         CALL  #MOV_Descarga
         ( Sensor_Pieza               := ,
           Sensor_Pinza_Llena         := ,
           Sensor_Llegada_a_Maquina   := ,
           Sensor_Llegada_a_Buffer    := ,
           "Sensor_Llegada_a _Reposo" := ,
           EMER                       := TRUE,
           Tiempo_lim                 := #Tiempo_lim,
           Timer_LIM                  := #Timer_LIM,
           MOV1                       := #Mov1,
           MOV2                       := #Mov2,
           MOV3                       := #Mov3,
           ACT1                       := #Act1,
           ACT2                       := #Act2,
           Aviso_Error_Tiempo_Limite  := #Aviso_Tiempo_Lim,
           Aviso_Fin_Maniobra         := #Aviso_Fin_Maniobra,
           Aviso_Error_No_Pieza       := #Aviso_No_Pieza,
           Aviso_Error_Pinza_Abierta  := #Aviso_Pinza_Abierta
         );



   _ERROR_ASINCRONO:NOP   0;
END_REGION

REGION Network 6: SALIDA ERROR SINCRONO
         A     #X_Error_Sincrono;
         AN    #Aviso_Error_Sincrono;
         S     #X_REPOSO;
         R     #X_Error_Sincrono;
END_REGION

REGION Network 7: SALIDA ERROR ASINCRONO
         A     #X_Error_Asincrono;
         AN    #Aviso_Error_Asincrono;
         S     #X_REPOSO;
         R     #X_Error_Asincrono;
END_REGION

REGION Network 8: START===TRUE
         A     #START;
         FP    #BDT;

         S     #X_REPOSO;
         R     #X_1_1;
         R     #X_1_2;
END_REGION

REGION Network 9: X_REPOSO--->X_1_1
   // Este modo se activa para el torno y la prensa
         A     #X_REPOSO;
         A     #X_Marcha_1;
         AN    #X_Marcha_2;
         A     #Sensor_Llegada_a_Reposo;
         A     #Sensor_Pieza;
         AN    #Sensor_Pinza_Llena;
         AN    #Sensor_Llegada_Carga;
         AN    #Sensor_Llegada_Descarga;


         S     #X_1_1;
         R     #X_REPOSO;
END_REGION

REGION Network 10: X_REPOSO--->X_1_2
   // Este modo se activa
         A     #X_REPOSO;
         A     #X_Marcha_2;
         AN    #X_Marcha_1;
         A     #Sensor_Llegada_a_Reposo;
         A     #Sensor_Pieza;  //si no hay pieza no llamo al bloque  NO UTILITY
         AN    #Sensor_Pinza_Llena;  //la pinza esta ocupada, no puede ir a por otra pieza
         AN    #Sensor_Llegada_Carga;
         AN    #Sensor_Llegada_Descarga;


         S     #X_1_2;
         R     #X_REPOSO;
END_REGION

REGION Network 11: X_1_1--->X_REPOSO
         A     #X_1_1;
         A     #Aviso_Fin_Maniobra;

         S     #X_REPOSO;
         R     #X_1_1;
         R     #Aviso_Fin_Maniobra;
END_REGION

REGION Network 12: X_1_2--->X_REPOSO
         A     #X_1_2;
         A     #Aviso_Fin_Maniobra;

         S     #X_REPOSO;
         R     #X_1_2;
         R     #Aviso_Fin_Maniobra;
END_REGION

REGION Network 13: TRAT X_REPOSO
         A     #X_REPOSO;
         =     #STDBY;
END_REGION

REGION Network 14: TRAT X_1_1
         A     #X_1_1;


         JCN   _MOV_1;

         CALL  #MOV_Carga
         ( Sensor_Pieza               := #Sensor_Pieza,
           Sensor_Pinza_Llena         := #Sensor_Pinza_Llena,
           Sensor_Llegada_a_Buffer    := #Sensor_Llegada_Carga,
           Sensor_Llegada_a_Maquina   := #Sensor_Llegada_Descarga,
           "Sensor_Llegada_a _Reposo" := #Sensor_Llegada_a_Reposo,
           EMER                       := FALSE,
           Tiempo_lim                 := #Tiempo_lim,
           Timer_LIM                  := #Timer_LIM,
           MOV1                       := #Mov1,
           MOV2                       := #Mov2,
           MOV3                       := #Mov3,
           ACT1                       := #Act1,
           ACT2                       := #Act2,
           WAIT1                      := #Wait,
           Aviso_Error_Tiempo_Limite  := #Aviso_Tiempo_Lim,
           Aviso_Fin_Maniobra         := #Aviso_Fin_Maniobra,
           Aviso_Error_No_Pieza       := #Aviso_No_Pieza,
           Aviso_Error_Pinza_Abierta  := #Aviso_Pinza_Abierta,
           Aviso_Maquina_Libre        := #Aviso_Maquina_Libre
         );


   _MOV_1:NOP   0;
END_REGION

REGION Network 15: TRAT X_1_2
         A     #X_1_2;

         JCN   _MOV_2;

         CALL  #MOV_Descarga
         ( Sensor_Pieza               := #Sensor_Pieza,
           Sensor_Pinza_Llena         := #Sensor_Pinza_Llena,
           Sensor_Llegada_a_Maquina   := #Sensor_Llegada_Carga,
           Sensor_Llegada_a_Buffer    := #Sensor_Llegada_Descarga,
           "Sensor_Llegada_a _Reposo" := #Sensor_Llegada_a_Reposo,
           EMER                       := FALSE,
           Tiempo_lim                 := #Tiempo_lim,
           Timer_LIM                  := #Timer_LIM,
           MOV1                       := #Mov1,
           MOV2                       := #Mov2,
           MOV3                       := #Mov3,
           ACT1                       := #Act1,
           ACT2                       := #Act2,
           Aviso_Error_Tiempo_Limite  := #Aviso_Tiempo_Lim,
           Aviso_Fin_Maniobra         := #Aviso_Fin_Maniobra,
           Aviso_Error_No_Pieza       := #Aviso_No_Pieza,
           Aviso_Error_Pinza_Abierta  := #Aviso_Pinza_Abierta
         );

   _MOV_2:NOP   0;
END_REGION
END_FUNCTION_BLOCK

// folder: metacontrol

FUNCTION "grafcet_modos_de_marcha" : Void   // FC1, LAD
TITLE = Grafcet que gestiona al menos 2 modos de marcha: A y B
{ S7_Optimized_Access := 'TRUE' }
VERSION : 0.1
// Modo A:  hace referencia a un subconjunto de los parámetros (DB4) de todos los parámetros (DB1)
// Modo B:  hace referencia a un subconjunto de los parámetros (DB5) de todos los parámetros (DB1)
// 
// Tratamiento del modo A: transferir el subconjunto de parámetros del modo A (DB4) a  DB1
// Tratamiento del modo B: transferir el subconjunto de parámetros del modo B (DB5) a  DB1
// (ver diapositiva 24 de "modos de marcha"- flexibilidad en producción (1/2))
// 
// Consideraciones generales: todo el código de producción tira de DB1. El tratamiento de cada modo es simplemente un paso de información entre bloques de datos. EL PROGRAMA DE CONTROL no se ve afectado.
BEGIN

REGION Network 1: Modo de marcha A
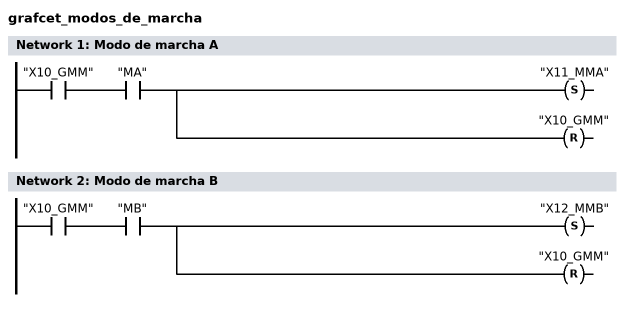
   RUNG wire#powerrail
      Contact( "X10_GMM" )
      Contact( "MA" )
      wire#w1
      S_Coil( "X11_MMA" )
   END_RUNG
   RUNG wire#w1
      R_Coil( "X10_GMM" )
   END_RUNG
   // the same network as SCL:
   IF "X10_GMM" AND "MA" THEN
       "X11_MMA" := TRUE;
       "X10_GMM" := FALSE;
   END_IF;
END_REGION

REGION Network 2: Modo de marcha B
   RUNG wire#powerrail
      Contact( "X10_GMM" )
      Contact( "MB" )
      wire#w1
      S_Coil( "X12_MMB" )
   END_RUNG
   RUNG wire#w1
      R_Coil( "X10_GMM" )
   END_RUNG
   // the same network as SCL:
   IF "X10_GMM" AND "MB" THEN
       "X12_MMB" := TRUE;
       "X10_GMM" := FALSE;
   END_IF;
END_REGION

REGION Network 3 (STL): Salida de MMA
         A     "X11_MMA";
         AN    "MA";
         S     "X10_GMM";
         R     "X11_MMA";
END_REGION

REGION Network 4 (STL): Salida de MMB
         A     "X12_MMB";
         AN    "MB";
         S     "X10_GMM";
         R     "X12_MMB";
END_REGION

REGION Network 5 (STL): Carga de valores para MA
   // Se van a mantener los valores de error en las distintas maniobras. Se cambia:
   // -El valor de la fuerza requerida en el Conformado
   // -La temperatura adecuada para poder empezar el proceso para el Horno y la Tunel
   // -El tiempo maximo en detectar un error en la acción de la Pulidora
         A     "X11_MMA";
         JCN   _carga_valores_modo_A;

         L     "DATOS_PRODUCCION_MODO_A".Fuerza_necesaria_CONFOR;
         T     "DATOS_PRODUCCION".Fuerza_necesaria_CONFOR;
   //fuerza a realizar en la prensa
         L     "DATOS_PRODUCCION_MODO_A".Temperatura_necesaria_HORNO;
         T     "DATOS_PRODUCCION".Temperatura_OK_HORNO;
   // temperatura alcanzada para funcionamiento horno
         L     "DATOS_PRODUCCION_MODO_A".Temperatura_necesaria_TUNEL;
         T     "DATOS_PRODUCCION".Temperatura_OK_TUNEL;
   // temperatura alcanzada para funcionamiento horno

         L     "DATOS_PRODUCCION_MODO_A".Tiempo_lim_PULIDO;
         T     "DATOS_PRODUCCION".T_PULI_Pulido;
   //tiempo limite de procesado
   _carga_valores_modo_A:NOP   0;
END_REGION

REGION Network 6 (STL): Carga de valores para MB
   // Se van a mantener los valores de error en las distintas maniobras. Se cambia:
   // -El valor de la fuerza requerida en el Conformado
   // -La temperatura adecuada para poder empezar el proceso para el Horno y la Tunel
   // -El tiempo maximo en detectar un error en la acción de la Pulidora
         A     "X12_MMB";
         JCN   _carga_valores_modo_B;

         L     "DATOS_PRODUCCION_MODO_B".Fuerza_necesaria_CONFOR;
         T     "DATOS_PRODUCCION".Fuerza_necesaria_CONFOR;
   //fuerza a realizar en la prensa
         L     "DATOS_PRODUCCION_MODO_B".Temperatura_necesaria_HORNO;
         T     "DATOS_PRODUCCION".Temperatura_OK_HORNO;
   // temperatura alcanzada para funcionamiento horno
         L     "DATOS_PRODUCCION_MODO_B".Temperatura_necesaria_TUNEL;
         T     "DATOS_PRODUCCION".Temperatura_OK_TUNEL;
   // temperatura alcanzada para funcionamiento horno

         L     "DATOS_PRODUCCION_MODO_B".Tiempo_lim_PULIDO;
         T     "DATOS_PRODUCCION".T_PULI_Pulido;
   //tiempo limite de procesado

   _carga_valores_modo_B:NOP   0;
END_REGION
END_FUNCTION

FUNCTION "grafcet_seguridad" : Void   // FC4, LAD
TITLE = grafcet para la gestión de parada brusca- paso a defecto seta EMER
{ S7_Optimized_Access := 'TRUE' }
VERSION : 0.1
// Gobierna los eventos asíncronos y (al menos) gestiona dos estados: Marcha y Defecto-
// Se coordina jerárquicamente (mediante FORZADO) con el resto de grafcets (modos_de_marcha y conjunto de grafcets de producción).
// (ver diapositivas- Modos de marcha).
// 
// Como consecuencia de la vuelta del defecto a producción (rearme):
// 1.Se debe informar a las máquinas de este hecho (a través del interfaz EMER de la plantilla de máquina). A su vez cada bloque máquina debe informar a sus maniobras.
// 2.Se debe informar al Grafcet/s de Producción y de modo_de_marcha que vuelvan a un estado de producción (por ejemplo el estado de reposo).
BEGIN

REGION Network 1 (STL): etapa de defecto global, activación de la seta de emergencia (GEMER)
         A     "EMER";
         S     "X21_EMER";
         R     "X20_Marcha";
END_REGION

REGION Network 2 (STL): tratamiento del defecto- forzado GP
   // Forzado- desconecta todos los estados de GP (no hay un estado de EMER en GP explícito)
         A     "X21_EMER";
         S     "X10_GMM";  //debe forzar al grafcet de modos de marcha
   //al ser un evento asíncrono debo resetear todos los estados
         R     "X1";
         R     "X2";
         R     "X3";
         R     "X4";
         R     "X5";
         R     "X_CONFORMADO";
         R     "X_HORNO";
         R     "X_TUNEL";
         R     "X_PULIDORA";
         R     "X_ROBOT";

         R     "X11_MMA";
         R     "X12_MMB";
END_REGION

REGION Network 3 (STL): tratamiento del defecto- llamadas a las máquinas informando de EMER
   // acciones de forzado sobre GP
         A     "X21_EMER";

         JCN   _forzado_maquinas;

         CALL  "CONFORMADORA", "CONFORMADORA_DB"
         ( START                    := "START_CONFOR",
           REARME                   := "Rearme_CONFOR",
           EMER                     := TRUE,
           S_fin                    := "S_final_CONFOR",
           Tiempo_MAX_maniobra      := "DATOS_PRODUCCION".Tiempo_lim_CONFOR,
           Temp_Ciclo_compre        := "T_compresion_CONFOR",
           Temp_Ciclo_descompre     := "T_descompresion_CONFOR",
           Fuerza_SENSOR            := "Fuerza_SENSOR_CONFOR",
           HI_LIM                   := "DATOS_PRODUCCION".HI_LIM,
           LO_LIM                   := "DATOS_PRODUCCION".LOW_LIM,
           Aviso_Pieza_Cargada      := "Aviso_Pieza_Cargada_CONFOR",
           Aviso_Pieza_Descargada   := "Aviso_Pieza_Desargada_CONFOR",
           FUERZA_NECESARIA         := "DATOS_PRODUCCION".Fuerza_necesaria_CONFOR,
           COMPRIMIR                := "COMPRIMIR_CONFOR",
           DESCOMPRIR               := "DESCOMPRIMIR_CONFOR",
           Aviso_Standby            := "Aviso_Standby_CONFOR",
           Aviso_error_sincrono_EXT := "Aviso_error_sincrono_EXT_CONFOR",
           Aviso_error_sensor_EXT   := "Aviso_error_sensor_EXT_CONFOR",
           FUERZA_REAL              := "Fuerza_REAL_CONFOR"
         );

         CALL  "maq_temp", "maq_temp_DB_HORNO"
         ( START                    := "START_HORNO",
           REARME                   := "Rearme_HORNO",
           EMER                     := TRUE,
           Tiempo_MAX_maniobra      := "DATOS_PRODUCCION".Tiempo_lim_Cinta_Horno,
           Tempo_maniobra           := "T_Cinta_Horno",
           Temperatura_SENSOR       := "Temperatura_SENSOR_HORNO",
           HI_LIM                   := "DATOS_PRODUCCION".HI_LIM,
           LO_LIM                   := "DATOS_PRODUCCION".LOW_LIM,
           Modo_Foco                := TRUE,
           Aviso_Piezas_Cargadas    := "S_piezas_cargadas_HORNO",
           Aviso_Piezas_Descargadas := "S_piezas_descargadas_HORNO",
           Temperatura_limite       := "DATOS_PRODUCCION".Temperatura_lim_HORNO,
           Temperatura_OK           := "DATOS_PRODUCCION".Temperatura_OK_HORNO,
           FOCO                     := "FOCO_HORNO",
           MOV                      := "MOV_CINTA_HORNO",
           Aviso_OK                 := "Aviso_Foco_OK_HORNO",
           Aviso_Standby            := "Aviso_Standby_HORNO",
           Aviso_error_sincrono_EXT := "Aviso_error_sincrono_EXT_HORNO",
           Aviso_error_sensor_EXT   := "Aviso_error_sensor_EXT_HORNO",
           Temperatura_REAL         := "Temperatura_REAL_HORNO"
         );

         CALL  "maq_temp","maq_temp_DB_TUNEL"
         ( START                    := "START_TUNEL",
           REARME                   := "Rearme_TUNEL",
           EMER                     := TRUE,
           Tiempo_MAX_maniobra      := "DATOS_PRODUCCION".Tiempo_lim_Cinta_Tunel,
           Tempo_maniobra           := "T_Cinta_Tunel",
           Temperatura_SENSOR       := "Temperatura_SENSOR_TUNEL",
           HI_LIM                   := "DATOS_PRODUCCION".HI_LIM,
           LO_LIM                   := "DATOS_PRODUCCION".LOW_LIM,
           Modo_Foco                := FALSE,
           Aviso_Piezas_Cargadas    := "S_piezas_cargadas_TUNEL",
           Aviso_Piezas_Descargadas := "S_piezas_descargadas_TUNEL",
           Temperatura_limite       := "DATOS_PRODUCCION".Temperatura_lim_TUNEL,
           Temperatura_OK           := "DATOS_PRODUCCION".Temperatura_OK_TUNEL,
           FOCO                     := "FOCO_TUNEL",
           MOV                      := "MOV_CINTA_TUNEL",
           Aviso_OK                 := "Aviso_Foco_OK_TUNEL",
           Aviso_Standby            := "Aviso_Standby_TUNEL",
           Aviso_error_sincrono_EXT := "Aviso_error_sincrono_EXT_TUNEL",
           Aviso_error_sensor_EXT   := "Aviso_error_sensor_EXT_TUNEL",
           Temperatura_REAL         := "Temperatura_REAL_TUNEL"
         );

         CALL  "PULIDORA", "PULIDORA_DB"
         ( Spieza                := "Spieza_PULI",
           SFMovCab              := "S_F_Mov_Cab",
           SFMovCab2             := "S_F_Mov_Cab2",
           SF_Acercar            := "S_F_Acercar",
           SFPulido1             := "S_F_Pulido1",
           SFPulido2             := "S_F_Pulido2",
           SFCambio              := "S_F_Cambio",
           SFAlejar              := "S_F_Alejar",
           SFGiro                := "S_F_Giro",
           SFGiro2               := "S_F_Giro2",
           T_Max_MovCab          := "DATOS_PRODUCCION".T_PULI_Pulido,
           T_Max_Mov_Cab2        := "DATOS_PRODUCCION".T_PULI_Pulido,
           T_Max_Acercar         := "DATOS_PRODUCCION".T_PULI_Mov_Puli,
           T_Max_Pulido          := "DATOS_PRODUCCION".T_PULI_Pulido,
           T_Max_Pulido2         := "DATOS_PRODUCCION".T_PULI_Pulido,
           T_Max_Cambio          := "DATOS_PRODUCCION".T_PULI_Cambio,
           T_Max_Alejar          := "DATOS_PRODUCCION".T_PULI_Mov_Puli,
           T_Max_Giro            := "DATOS_PRODUCCION".T_PULI_Giro,
           T_Max_Giro2           := "DATOS_PRODUCCION".T_PULI_Giro,
           TMovCab               := "T_Mov_Cab",
           TMovCab2              := "T_Mov_Cab2",
           TAcercar              := "T_Acercar",
           TPulido1              := "T_Pulido1",
           TPulido2              := "T_Pulido2",
           TCambio               := "T_Cambio",
           TAlejar               := "T_Alejar",
           TGiro                 := "T_Giro",
           TGiro2                := "T_Giro2",
           START                 := "START_PULI",
           REARME                := "REARME_PULI",
           EMER                  := TRUE,
           Mover_Cabezal         := "Mover_Cabezal1",
           Mover_Cabezal2        := "Mover_Cabezal2",
           Acercar_              := "Acercar",
           Pulido_               := "Pulido1",
           Cambio_               := "Cambio",
           Pulido2_              := "Pulido2",
           Alejar_               := "Alejar",
           Giro_                 := "Giro_Soporte1",
           Giro2                 := "Giro_Soporte2",
           Aviso_StandBy         := "Aviso_StdBy_PULI",
           Aviso_Error_Asíncrono := "Aviso_Error_Asinc_PULI",
           Aviso_Error_Sincrono  := "Aviso_Error_Sinc_PULI"
         );

         CALL  "ROBOT", "ROBOT_DB"
         ( Sensor_Pieza            := "SB_pieza_esperando",
           Sensor_Pinza_Llena      := "SB_pinza_llena_brazo",
           Sensor_Llegada_Carga    := "SB_llegada_Carga",
           Sensor_Llegada_Descarga := "SB_llegada_Descarga",
           Sensor_Llegada_a_Reposo := "SB_llegada_a_reposo",
           START                   := "START_ROBOT",
           EMER                    := TRUE,
           REARME                  := "Rearme_ROBOT",
           Tiempo_lim              := "DATOS_PRODUCCION".Tiempo_lim_brazo,
           Timer_LIM               := "Tlimite_ROBOT",
           X_Marcha_1              := "MODO_M1_Descarga_ROBOT",
           X_Marcha_2              := "MODO_M2_Carga_ROBOT",
           Mov1                    := "Mov1",
           Mov2                    := "Mov2",
           Mov3                    := "Mov3",
           Act1                    := "Act1",
           Act2                    := "Act2",
           Wait                    := "X_Espera_maquina_libre",
           Aviso_Emergencia        := "Aviso_emergencia_ROBOT",
           STDBY                   := "Aviso_STDBY_ROBOT",
           Aviso_Maquina_Libre     := "Aviso_maquina_libre",
           Aviso_Error_Sincrono    := "Aviso_error_sincrono_ROBOT",
           Aviso_Error_Asincrono   := "Aviso_error_asincrono_ROBOT"
         );

   _forzado_maquinas:NOP   0;
END_REGION

REGION Network 4 (STL): vuelta a funcionamiento desde defecto- se informa a las máquinas y se fuerza a GP a volver a producción
         A     "X21_EMER";
         AN    "EMER";
         A     "Rearme";

         JCN   _aviso_a_maquinas;

         CALL  "CONFORMADORA", "CONFORMADORA_DB"
         ( START                    := "START_CONFOR",
           REARME                   := TRUE,
           EMER                     := FALSE,
           S_fin                    := "S_final_CONFOR",
           Tiempo_MAX_maniobra      := "DATOS_PRODUCCION".Tiempo_lim_CONFOR,
           Temp_Ciclo_compre        := "T_compresion_CONFOR",
           Temp_Ciclo_descompre     := "T_descompresion_CONFOR",
           Fuerza_SENSOR            := "Fuerza_SENSOR_CONFOR",
           HI_LIM                   := "DATOS_PRODUCCION".HI_LIM,
           LO_LIM                   := "DATOS_PRODUCCION".LOW_LIM,
           Aviso_Pieza_Cargada      := "Aviso_Pieza_Cargada_CONFOR",
           Aviso_Pieza_Descargada   := "Aviso_Pieza_Desargada_CONFOR",
           FUERZA_NECESARIA         := "DATOS_PRODUCCION".Fuerza_necesaria_CONFOR,
           COMPRIMIR                := "COMPRIMIR_CONFOR",
           DESCOMPRIR               := "DESCOMPRIMIR_CONFOR",
           Aviso_Standby            := "Aviso_Standby_CONFOR",
           Aviso_error_sincrono_EXT := "Aviso_error_sincrono_EXT_CONFOR",
           Aviso_error_sensor_EXT   := "Aviso_error_sensor_EXT_CONFOR",
           FUERZA_REAL              := "Fuerza_REAL_CONFOR"
         );

         CALL  "maq_temp", "maq_temp_DB_HORNO"
         ( START                    := "START_HORNO",
           REARME                   := TRUE,
           EMER                     := FALSE,
           Tiempo_MAX_maniobra      := "DATOS_PRODUCCION".Tiempo_lim_Cinta_Horno,
           Tempo_maniobra           := "T_Cinta_Horno",
           Temperatura_SENSOR       := "Temperatura_SENSOR_HORNO",
           HI_LIM                   := "DATOS_PRODUCCION".HI_LIM,
           LO_LIM                   := "DATOS_PRODUCCION".LOW_LIM,
           Modo_Foco                := TRUE,
           Aviso_Piezas_Cargadas    := "S_piezas_cargadas_HORNO",
           Aviso_Piezas_Descargadas := "S_piezas_descargadas_HORNO",
           Temperatura_limite       := "DATOS_PRODUCCION".Temperatura_lim_HORNO,
           Temperatura_OK           := "DATOS_PRODUCCION".Temperatura_OK_HORNO,
           FOCO                     := "FOCO_HORNO",
           MOV                      := "MOV_CINTA_HORNO",
           Aviso_OK                 := "Aviso_Foco_OK_HORNO",
           Aviso_Standby            := "Aviso_Standby_HORNO",
           Aviso_error_sincrono_EXT := "Aviso_error_sincrono_EXT_HORNO",
           Aviso_error_sensor_EXT   := "Aviso_error_sensor_EXT_HORNO",
           Temperatura_REAL         := "Temperatura_REAL_HORNO"
         );

         CALL  "maq_temp","maq_temp_DB_TUNEL"
         ( START                    := "START_TUNEL",
           REARME                   := TRUE,
           EMER                     := FALSE,
           Tiempo_MAX_maniobra      := "DATOS_PRODUCCION".Tiempo_lim_Cinta_Tunel,
           Tempo_maniobra           := "T_Cinta_Tunel",
           Temperatura_SENSOR       := "Temperatura_SENSOR_TUNEL",
           HI_LIM                   := "DATOS_PRODUCCION".HI_LIM,
           LO_LIM                   := "DATOS_PRODUCCION".LOW_LIM,
           Modo_Foco                := FALSE,
           Aviso_Piezas_Cargadas    := "S_piezas_cargadas_TUNEL",
           Aviso_Piezas_Descargadas := "S_piezas_descargadas_TUNEL",
           Temperatura_limite       := "DATOS_PRODUCCION".Temperatura_lim_TUNEL,
           Temperatura_OK           := "DATOS_PRODUCCION".Temperatura_OK_TUNEL,
           FOCO                     := "FOCO_TUNEL",
           MOV                      := "MOV_CINTA_TUNEL",
           Aviso_OK                 := "Aviso_Foco_OK_TUNEL",
           Aviso_Standby            := "Aviso_Standby_TUNEL",
           Aviso_error_sincrono_EXT := "Aviso_error_sincrono_EXT_TUNEL",
           Aviso_error_sensor_EXT   := "Aviso_error_sensor_EXT_TUNEL",
           Temperatura_REAL         := "Temperatura_REAL_TUNEL"
         );

         CALL  "PULIDORA", "PULIDORA_DB"
         ( Spieza                := "Spieza_PULI",
           SFMovCab              := "S_F_Mov_Cab",
           SFMovCab2             := "S_F_Mov_Cab2",
           SF_Acercar            := "S_F_Acercar",
           SFPulido1             := "S_F_Pulido1",
           SFPulido2             := "S_F_Pulido2",
           SFCambio              := "S_F_Cambio",
           SFAlejar              := "S_F_Alejar",
           SFGiro                := "S_F_Giro",
           SFGiro2               := "S_F_Giro2",
           T_Max_MovCab          := "DATOS_PRODUCCION".T_PULI_Pulido,
           T_Max_Mov_Cab2        := "DATOS_PRODUCCION".T_PULI_Pulido,
           T_Max_Acercar         := "DATOS_PRODUCCION".T_PULI_Mov_Puli,
           T_Max_Pulido          := "DATOS_PRODUCCION".T_PULI_Pulido,
           T_Max_Pulido2         := "DATOS_PRODUCCION".T_PULI_Pulido,
           T_Max_Cambio          := "DATOS_PRODUCCION".T_PULI_Cambio,
           T_Max_Alejar          := "DATOS_PRODUCCION".T_PULI_Mov_Puli,
           T_Max_Giro            := "DATOS_PRODUCCION".T_PULI_Giro,
           T_Max_Giro2           := "DATOS_PRODUCCION".T_PULI_Giro,
           TMovCab               := "T_Mov_Cab",
           TMovCab2              := "T_Mov_Cab2",
           TAcercar              := "T_Acercar",
           TPulido1              := "T_Pulido1",
           TPulido2              := "T_Pulido2",
           TCambio               := "T_Cambio",
           TAlejar               := "T_Alejar",
           TGiro                 := "T_Giro",
           TGiro2                := "T_Giro2",
           START                 := "START_PULI",
           REARME                := TRUE,
           EMER                  := FALSE,
           Mover_Cabezal         := "Mover_Cabezal1",
           Mover_Cabezal2        := "Mover_Cabezal2",
           Acercar_              := "Acercar",
           Pulido_               := "Pulido1",
           Cambio_               := "Cambio",
           Pulido2_              := "Pulido2",
           Alejar_               := "Alejar",
           Giro_                 := "Giro_Soporte1",
           Giro2                 := "Giro_Soporte2",
           Aviso_StandBy         := "Aviso_StdBy_PULI",
           Aviso_Error_Asíncrono := "Aviso_Error_Asinc_PULI",
           Aviso_Error_Sincrono  := "Aviso_Error_Sinc_PULI"
         );

         CALL  "ROBOT", "ROBOT_DB"
         ( Sensor_Pieza            := "SB_pieza_esperando",
           Sensor_Pinza_Llena      := "SB_pinza_llena_brazo",
           Sensor_Llegada_Carga    := "SB_llegada_Carga",
           Sensor_Llegada_Descarga := "SB_llegada_Descarga",
           Sensor_Llegada_a_Reposo := "SB_llegada_a_reposo",
           START                   := "START_ROBOT",
           EMER                    := FALSE,
           REARME                  := TRUE,
           Tiempo_lim              := "DATOS_PRODUCCION".Tiempo_lim_brazo,
           Timer_LIM               := "Tlimite_ROBOT",
           X_Marcha_1              := "MODO_M1_Descarga_ROBOT",
           X_Marcha_2              := "MODO_M2_Carga_ROBOT",
           Mov1                    := "Mov1",
           Mov2                    := "Mov2",
           Mov3                    := "Mov3",
           Act1                    := "Act1",
           Act2                    := "Act2",
           Wait                    := "X_Espera_maquina_libre",
           Aviso_Emergencia        := "Aviso_emergencia_ROBOT",
           STDBY                   := "Aviso_STDBY_ROBOT",
           Aviso_Maquina_Libre     := "Aviso_maquina_libre",
           Aviso_Error_Sincrono    := "Aviso_error_sincrono_ROBOT",
           Aviso_Error_Asincrono   := "Aviso_error_asincrono_ROBOT"
         );


   _aviso_a_maquinas:NOP   0;

         A     "X21_EMER";
         AN    "EMER";
         A     "Rearme";
         S     "X20_Marcha";
         S     "X0";
         R     "X21_EMER";
END_REGION
END_FUNCTION

// folder: tests

FUNCTION "test_trat_sensor_temperatura" : Void   // FC3, STL
{ S7_Optimized_Access := 'TRUE' }
VERSION : 0.1
BEGIN

REGION Network 1: CALL a TRAT_SENSOR_TEMPERATURA
   // En este bloque se comprueba si el funcionamiento de la temperatura para HORNO y TUNEL
         CALL  "TRAT_SENSOR_TEMPERATURA"
         ( RAW                  := "Temperatura_SENSOR_HORNO",
           BIPOLAR              := FALSE,
           HI_LIM               := 1000.0,
           LO_LIM               := 0.0,
           Temperatura_limite   := 800.0,
           Temperatura_OK       := 600.0,
           Modo_FOCO            := TRUE,
           RESET                := FALSE,
           Aviso_Foco_encendido := "FOCO_HORNO",
           Aviso_Foco_OK        := "Aviso_Foco_OK_HORNO",
           Error                := "Aviso_Error_Sinc_PULI",
           Real_Val             := "Temperatura_REAL_HORNO"
         );

         CALL  "TRAT_SENSOR_TEMPERATURA"
         ( RAW                  := "Temperatura_SENSOR_HORNO",
           BIPOLAR              := FALSE,
           HI_LIM               := 1000.0,
           LO_LIM               := 0.0,
           Temperatura_limite   := 600.0,
           Temperatura_OK       := 800.0,
           Modo_FOCO            := FALSE,
           RESET                := FALSE,
           Aviso_Foco_encendido := "FOCO_TUNEL",
           Aviso_Foco_OK        := "Aviso_Foco_OK_HORNO",
           Error                := "Aviso_Error_Sinc_PULI",
           Real_Val             := "Temperatura_REAL_HORNO"
         );
END_REGION
END_FUNCTION

FUNCTION "test_COMFORMADORA" : Void   // FC5, STL
TITLE = TEST del maquina COMFORMADORA
{ S7_Optimized_Access := 'TRUE' }
VERSION : 0.1
BEGIN

REGION Network 1: CALL CONFORMADORA

         CALL  "CONFORMADORA", "CONFORMADORA_DB"
         ( START                    := "START_CONFOR",
           REARME                   := "Rearme_CONFOR",
           EMER                     := "Emer_CONFOR",
           S_fin                    := "S_final_CONFOR",
           Tiempo_MAX_maniobra      := "DATOS_PRODUCCION".Tiempo_lim_CONFOR,
           Temp_Ciclo_compre        := "T_compresion_CONFOR",
           Temp_Ciclo_descompre     := "T_descompresion_CONFOR",
           Fuerza_SENSOR            := "Fuerza_SENSOR_CONFOR",
           HI_LIM                   := 1000.0,
           LO_LIM                   := 0.0,
           Aviso_Pieza_Cargada      := "Aviso_Pieza_Cargada_CONFOR",
           Aviso_Pieza_Descargada   := "Aviso_Pieza_Desargada_CONFOR",
           FUERZA_NECESARIA         := 600.0,
           COMPRIMIR                := "COMPRIMIR_CONFOR",
           DESCOMPRIR               := "DESCOMPRIMIR_CONFOR",
           Aviso_Standby            := "Aviso_Standby_CONFOR",
           Aviso_error_sincrono_EXT := "Aviso_error_sincrono_EXT_CONFOR",
           Aviso_error_sensor_EXT   := "Aviso_error_sensor_EXT_CONFOR",
           FUERZA_REAL              := "Fuerza_REAL_CONFOR"
         );
END_REGION
END_FUNCTION

FUNCTION "test_maq_temp" : Void   // FC6, STL
TITLE = TEST de las maquinas de control de temperatura
{ S7_Optimized_Access := 'TRUE' }
VERSION : 0.1
// Se hace un call al bloque FB y te utilizan distintos bloques de datos para consolidar la maquina de horno de sinterizado y tunel de secado
BEGIN

REGION Network 1: CALL HORNO / TUNEL

         CALL  "maq_temp", "maq_temp_DB_HORNO"
         ( START                    := "START_HORNO",
           REARME                   := "Rearme_HORNO",
           EMER                     := "Emer_HORNO",
           Tiempo_MAX_maniobra      := "DATOS_PRODUCCION".Tiempo_lim_Cinta_Horno,
           Tempo_maniobra           := "T_Cinta_Horno",
           Temperatura_SENSOR       := "Temperatura_SENSOR_HORNO",
           HI_LIM                   := 1000.0,
           LO_LIM                   := 0.0,
           Modo_Foco                := TRUE,
           Aviso_Piezas_Cargadas    := "S_piezas_cargadas_HORNO",
           Aviso_Piezas_Descargadas := "S_piezas_descargadas_HORNO",
           Temperatura_limite       := 800.0,
           Temperatura_OK           := 600.0,
           FOCO                     := "FOCO_HORNO",
           MOV                      := "MOV_CINTA_HORNO",
           Aviso_OK                 := "Aviso_Foco_OK_HORNO",
           Aviso_Standby            := "Aviso_Standby_HORNO",
           Aviso_error_sincrono_EXT := "Aviso_error_sincrono_EXT_HORNO",
           Aviso_error_sensor_EXT   := "Aviso_error_sensor_EXT_HORNO",
           Temperatura_REAL         := "Temperatura_REAL_HORNO"
         );

         CALL  "maq_temp","maq_temp_DB_TUNEL"
         ( START                    := "START_TUNEL",
           REARME                   := "Rearme_TUNEL",
           EMER                     := "Emer_TUNEL",
           Tiempo_MAX_maniobra      := "DATOS_PRODUCCION".Tiempo_lim_Cinta_Tunel,
           Tempo_maniobra           := "T_Cinta_Tunel",
           Temperatura_SENSOR       := "Temperatura_SENSOR_TUNEL",
           HI_LIM                   := 1000.0,
           LO_LIM                   := 0.0,
           Modo_Foco                := FALSE,
           Aviso_Piezas_Cargadas    := "S_piezas_cargadas_TUNEL",
           Aviso_Piezas_Descargadas := "S_piezas_descargadas_TUNEL",
           Temperatura_limite       := 5.0,
           Temperatura_OK           := 0.0,
           FOCO                     := "FOCO_TUNEL",
           MOV                      := "MOV_CINTA_TUNEL",
           Aviso_OK                 := "Aviso_Foco_OK_TUNEL",
           Aviso_Standby            := "Aviso_Standby_TUNEL",
           Aviso_error_sincrono_EXT := "Aviso_error_sincrono_EXT_TUNEL",
           Aviso_error_sensor_EXT   := "Aviso_error_sensor_EXT_TUNEL",
           Temperatura_REAL         := "Temperatura_REAL_TUNEL"
         );
END_REGION
END_FUNCTION

FUNCTION "test_PULIDORA" : Void   // FC7, STL
TITLE = TEST de la maquina PULIDORA
{ S7_Optimized_Access := 'TRUE' }
VERSION : 0.1
BEGIN

REGION Network 1: CALL PULIDORA
         CALL  "PULIDORA", "PULIDORA_DB"
         ( Spieza                := "Spieza_PULI",
           SFMovCab              := "S_F_Mov_Cab",
           SFMovCab2             := "S_F_Mov_Cab2",
           SF_Acercar            := "S_F_Acercar",
           SFPulido1             := "S_F_Pulido1",
           SFPulido2             := "S_F_Pulido2",
           SFCambio              := "S_F_Cambio",
           SFAlejar              := "S_F_Alejar",
           SFGiro                := "S_F_Giro",
           SFGiro2               := "S_F_Giro2",
           T_Max_MovCab          := "DATOS_PRODUCCION".T_PULI_Pulido,
           T_Max_Mov_Cab2        := "DATOS_PRODUCCION".T_PULI_Pulido,
           T_Max_Acercar         := "DATOS_PRODUCCION".T_PULI_Mov_Puli,
           T_Max_Pulido          := "DATOS_PRODUCCION".T_PULI_Pulido,
           T_Max_Pulido2         := "DATOS_PRODUCCION".T_PULI_Pulido,
           T_Max_Cambio          := "DATOS_PRODUCCION".T_PULI_Cambio,
           T_Max_Alejar          := "DATOS_PRODUCCION".T_PULI_Mov_Puli,
           T_Max_Giro            := "DATOS_PRODUCCION".T_PULI_Giro,
           T_Max_Giro2           := "DATOS_PRODUCCION".T_PULI_Giro,
           TMovCab               := "T_Mov_Cab",
           TMovCab2              := "T_Mov_Cab2",
           TAcercar              := "T_Acercar",
           TPulido1              := "T_Pulido1",
           TPulido2              := "T_Pulido2",
           TCambio               := "T_Cambio",
           TAlejar               := "T_Alejar",
           TGiro                 := "T_Giro",
           TGiro2                := "T_Giro2",
           START                 := "START_PULI",
           REARME                := "REARME_PULI",
           EMER                  := "EMER_PULI",
           Mover_Cabezal         := "Mover_Cabezal1",
           Mover_Cabezal2        := "Mover_Cabezal2",
           Acercar_              := "Acercar",
           Pulido_               := "Pulido1",
           Cambio_               := "Cambio",
           Pulido2_              := "Pulido2",
           Alejar_               := "Alejar",
           Giro_                 := "Giro_Soporte1",
           Giro2                 := "Giro_Soporte2",
           Aviso_StandBy         := "Aviso_StdBy_PULI",
           Aviso_Error_Asíncrono := "Aviso_Error_Asinc_PULI",
           Aviso_Error_Sincrono  := "Aviso_Error_Sinc_PULI"
         );
END_REGION
END_FUNCTION

FUNCTION "test_ROBOT" : Void   // FC9, STL
TITLE = TEST a bloque de ROBOT
{ S7_Optimized_Access := 'TRUE' }
VERSION : 0.1
BEGIN

REGION Network 1: CALL ROBOT

         CALL  "ROBOT", "ROBOT_DB"
         ( Sensor_Pieza            := "SB_pieza_esperando",
           Sensor_Pinza_Llena      := "SB_pinza_llena_brazo",
           Sensor_Llegada_Carga    := "SB_llegada_Carga",
           Sensor_Llegada_Descarga := "SB_llegada_Descarga",
           Sensor_Llegada_a_Reposo := "SB_llegada_a_reposo",
           START                   := "START_ROBOT",
           EMER                    := "EMER_ROBOT",
           REARME                  := "Rearme_ROBOT",
           Tiempo_lim              := "DATOS_PRODUCCION".Tiempo_lim_brazo,
           Timer_LIM               := "Tlimite_ROBOT",
           X_Marcha_1              := "MODO_M1_Descarga_ROBOT",
           X_Marcha_2              := "MODO_M2_Carga_ROBOT",
           Mov1                    := "Mov1",
           Mov2                    := "Mov2",
           Mov3                    := "Mov3",
           Act1                    := "Act1",
           Act2                    := "Act2",
           Wait                    := "X_Espera_maquina_libre",
           Aviso_Emergencia        := "Aviso_emergencia_ROBOT",
           STDBY                   := "Aviso_STDBY_ROBOT",
           Aviso_Maquina_Libre     := "Aviso_maquina_libre",
           Aviso_Error_Sincrono    := "Aviso_error_sincrono_ROBOT",
           Aviso_Error_Asincrono   := "Aviso_error_asincrono_ROBOT"
         );
END_REGION
END_FUNCTION